FUNCTION_BLOCK FB_ModeStateToColour
VAR_INPUT
	iModeState:INT;
END_VAR
VAR
END_VAR

VAR_OUTPUT
	qBackColour:DWORD;
	qTextColour:DWORD;
END_VAR

//theme:V5e09AHRtmc

//converts mode state as integer to colour as DWORD
CASE iModeState OF
	//0 = No State
	0:
	qBackColour := HMIColour.colourWhite;
	qTextColour	:= HMIColour.colourBlack;
	
	//1 = Power OFF	
	1:
	qBackColour := HMIColour.colourWhite;
	qTextColour	:= HMIColour.colourBlack;
	
	//2 = Power ON
	2:
	qBackColour := HMIColour.colourBlue;
	qTextColour	:= HMIColour.colourWhite;
	
	//3 = ManualMode
	3:
	qBackColour := HMIColour.colourBlue;
	qTextColour	:= HMIColour.colourWhite;
	
	//4 = AutoMode
	4:
	qBackColour := HMIColour.colourBlue;
	qTextColour	:= HMIColour.colourWhite;
	
	//5 = AutoCycling
	5:
	qBackColour := HMIColour.colourGreen;
	qTextColour	:= HMIColour.colourBlack;
	
	//6 = SemiAuto
	6:
	qBackColour := HMIColour.colourBlue;
	qTextColour	:= HMIColour.colourWhite;
	
	//7 = Fault
	7:
	qBackColour := HMIColour.colourRed;
	qTextColour	:= HMIColour.colourWhite;
	
	//8 = Bypass
	8:
	qBackColour := HMIColour.colourBlue;
	qTextColour	:= HMIColour.colourWhite;
	
	//9 = AutoCycleStopping
	9:
	qBackColour := HMIColour.colourGreen;
	qTextColour	:= HMIColour.colourBlack;
	
	//10 = Dry Cycle
	10:
	qBackColour := HMIColour.colourYellow;
	qTextColour	:= HMIColour.colourBlack;
	
	//11> = spare
	11..32767:
	qBackColour := HMIColour.colourWhite;
	qTextColour	:= HMIColour.colourBlack;
END_CASE

END_FUNCTION_BLOCK

(* stored: Version 1.1.0.1, ProductVersion 3.1.4024.12
   POU FB_ModeStateToColour: Id {7bb523b7-3f37-40a3-a2e4-99638f172644}, SpecialFunc None *)
